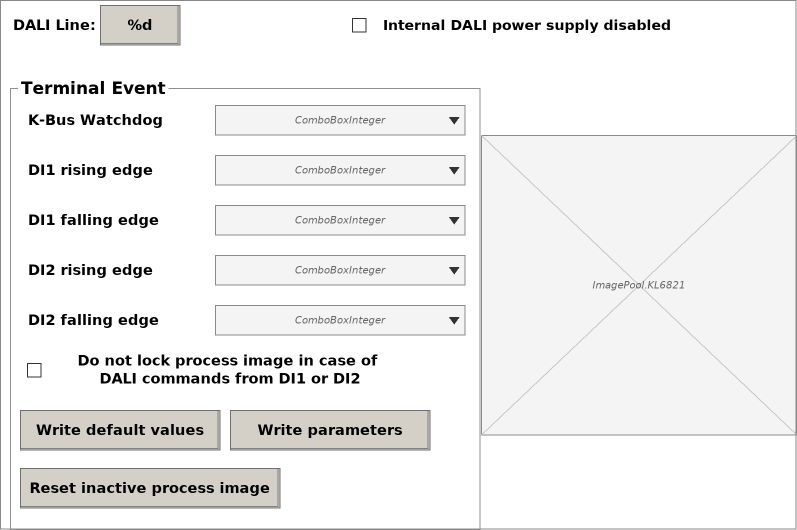
VISUALIZATION Visu_KL6821Configuration  // 797x530
    GroupBox (10,80 470x450), "Terminal Event"
        Textfield (15,25 170x30), "K-Bus Watchdog"
        ComboBoxInteger (205,25 250x30), variable: Communication.eCommandKBusWatchdog, text list: 'CommandOnTerminalEvent'
        Textfield (15,75 170x30), "DI1 rising edge"
        Textfield (15,125 170x30), "DI1 falling edge"
        ComboBoxInteger (205,75 250x30), variable: Communication.eCommandDI1RisingEdge, text list: 'CommandOnTerminalEvent'
        ComboBoxInteger (205,125 250x30), variable: Communication.eCommandDI1FallingEdge, text list: 'CommandOnTerminalEvent'
        Textfield (15,175 170x30), "DI2 rising edge"
        ComboBoxInteger (205,175 250x30), variable: Communication.eCommandDI2RisingEdge, text list: 'CommandOnTerminalEvent'
        Textfield (15,225 170x30), "DI2 falling edge"
        ComboBoxInteger (205,225 250x30), variable: Communication.eCommandDI2FallingEdge, text list: 'CommandOnTerminalEvent'
        Button (220,330 200x40), "Write parameters"
            OnMouseClick: execute { Communication.bInitialize := TRUE; }
        Button (10,330 200x40), "Write default values"
            OnMouseClick: execute { Communication.bDefaultValues := TRUE; }
        Button (10,388 260x40), "Reset inactive process image"
            OnMouseClick: execute { Communication.bResetInactiveProcessImage := TRUE; }
        Checkbox (15,275 35x30), variable: Communication.bDoNotLockProcessImage
        Textfield (50,267 340x45), "Do not lock process image in case of DALI commands from DI1 or DI2"
    Image (481,135 316x300), image: ImagePool.KL6821
    Group (350,10 330x30)
        Checkbox (0,0 34x30), variable: Communication.bInternalPowerSupplyDisabled
        Textfield (30,0 294x30), "Internal DALI power supply disabled"
    Group (10,5 170x40)
        Textfield (0,0 110x40), "DALI Line:"
        Button (90,0 80x40), "%d", text variable: GVL_Internal.nDALILine
            OnMouseClick: write the text variable via Default, min 1, max GVL_Internal.nNumberOfDALI_Lines, title "Choose line"
END_VISUALIZATION

(* stored: Version 1.1.0.1, ProductVersion 3.1.4024.12
   Visu Visu_KL6821Configuration: Id {41957b42-67f5-40cf-b8ac-5330d8fbfeea} *)
